FUNCTION_BLOCK MockEventHandler IMPLEMENTS I_EventHandler
VAR
	_eventsHandled : INT;
	lastEventHandled : I_Event;
END_VAR

METHOD PUBLIC EqualsLastEvent : bool
VAR_INPUT
	Event : I_Event;
END_VAR
EqualsLastEvent := lastEventHandled = Event;
END_METHOD

PROPERTY EventsHandled : int
GET
EventsHandled := _eventsHandled;
END_GET
END_PROPERTY

METHOD HandleEvent
VAR_INPUT
	Event	: I_Event;
END_VAR
_eventsHandled := _eventsHandled + 1;
lastEventHandled := Event;
END_METHOD

END_FUNCTION_BLOCK

(* stored: Version 1.1.0.1, ProductVersion 3.1.4024.12
   POU MockEventHandler: Id {58a62b4e-121a-499d-9f9c-e292ae4280ba}, SpecialFunc None
   Method EqualsLastEvent: Id {ea7149d7-32c0-463c-84fe-7104d0490fbd}
   Property EventsHandled: Id {ffaf055a-5ff2-4cf4-9302-3d63054b5abf}
   Get Get: Id {581825b6-ffe5-426e-ab27-85efbc5d8312}
   Method HandleEvent: Id {638fbefe-5ea6-4f53-b032-9046544ae9f1} *)
